// TIA Portal V17 export
// export: Created 2023-05-07T12:12:22.8691154Z, ExportSetting WithDefaults, DisplayName Totally Integrated Automation Portal, DisplayVersion V17, DisplayName TIA Portal Openness, DisplayVersion V17, DisplayName TIA Portal Version Control Interface, DisplayVersion V17, DisplayName TIA Portal Test Suite Advanced, DisplayVersion V17, DisplayName STEP 7 Professional, DisplayVersion V17, DisplayName SIMATIC Energy Suite, DisplayVersion V17, DisplayName STEP 7 Safety, DisplayVersion V17, DisplayName WinCC Professional, DisplayVersion V17
DATA_BLOCK "IMC+PID_DB"   // DB15
VERSION : 0.1
// stored: AutoNumber true, InstanceOfName IMC+PID, InstanceOfType FB
"IMC+PID"
   // VAR_INPUT
   //    SP : Real;
   //    PV : Real;
   // END_VAR
   // VAR_OUTPUT
   //    MV : Real;
   // END_VAR
   // VAR
   //    PV_model : Real;
   //    e_ob_mo : Real;
   //    "e" : Real;
   //    ef : Array[0..1] of Real;
   //    MV1 : Real;
   //    MV2 : Real;
   // END_VAR
BEGIN
END_DATA_BLOCK
